TYPE PuckData :
STRUCT
	RFID: DINT;
	Status: cPuckStatusEval;
	Device: DeviceData;
	PuckOnlyRoute: STRING(30);
	Side: STRING(30);
	IsCleaningEligible: BOOL;
END_STRUCT
END_TYPE

(* stored: Version 1.1.0.1, ProductVersion 3.1.4024.6
   DUT PuckData: Id {e2462ab7-ef85-4239-9a93-b9475b96c4b1} *)
